FUNCTION_BLOCK POU
VAR_INPUT
END_VAR
VAR_OUTPUT
END_VAR
VAR
	a: INT;
	b: INT;
END_VAR

a := a+b;

END_FUNCTION_BLOCK

(* stored: Version 1.1.0.1, ProductVersion 3.1.4024.13
   POU POU: Id {d708b816-d3ce-421d-8600-0c94f5ebf70b}, SpecialFunc None *)
